FUNCTION_BLOCK F_SEL_UINT_E_4 (* selection event-based selection) *)
  (* Standard: 61131-3; Classification: standard selection function; Description: Copyright (c) 2012 TU Wien ACIN This program and the accompanying materials are made available under the terms of the Eclipse Public License 2.0 which is available at https://www.eclipse.org/legal/epl-2.0/ SPDX-License-Identifier: EPL-2.0 *)
  (* Version 1.0, 2012-03-25, Monika Wenger, TU Wien ACIN *)
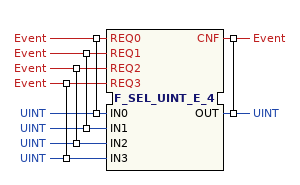
  EVENT_INPUT
    REQ0 WITH IN0;
    REQ1 WITH IN1;
    REQ2 WITH IN2;
    REQ3 WITH IN3;
  END_EVENT
  EVENT_OUTPUT
    CNF WITH OUT; (* Confirmation of Requested Service *)
  END_EVENT
  VAR_INPUT
    IN0 : UINT; (* Selectable input variable *)
    IN1 : UINT; (* Selectable input variable *)
    IN2 : UINT; (* Selectable input variable *)
    IN3 : UINT; (* Selectable input variable *)
  END_VAR
  VAR_OUTPUT
    OUT : UINT; (* Selected input *)
  END_VAR
END_FUNCTION_BLOCK
